// TIA Portal V17 export
// export: Created 2022-07-28T18:03:17.6934733Z, ExportSetting None, DisplayName Totally Integrated Automation Portal, DisplayVersion V17, DisplayName TIA Portal Openness, DisplayVersion V17, DisplayName TIA Portal Teamcenter Gateway, DisplayVersion V17, DisplayName TIA Portal Version Control Interface, DisplayVersion V17, DisplayName TIA Portal Test Suite Advanced, DisplayVersion V17, DisplayName SINAMICS Startdrive Advanced, DisplayVersion V17, DisplayName SINAMICS DCC, DisplayVersion V17, DisplayName SINAMICS Startdrive G130, G150, S120, S150, SINAMICS MV, S210, DisplayVersion V17, DisplayName SINAMICS Startdrive G110M, G120, G120C, G120D, G120P, G115D, DisplayVersion V17, DisplayName STEP 7 Professional, DisplayVersion V17, DisplayName SIMATIC Energy Suite, DisplayVersion V17, DisplayName STEP 7 CFC, DisplayVersion V17, DisplayName STEP 7 Safety, DisplayVersion V17, DisplayName WinCC Advanced / Unified PC, DisplayVersion V17, DisplayName SIMATIC Visualization Architect, DisplayVersion V17
TYPE "Lib_UDT_Int"
   STRUCT
      Tmp : Bool;   // Temp bool Var
      i_Tmp : Int;   // Temp Int Var
      r_Tmp : Real;   // Temp Real Var
      w_Tmp : Word;   // Temp Word Var
      dw_Tmp : DWord;   // Temp Dword Var
      di_Tmp : DInt;   // Temp DInt Var
      AlwTrue : Bool := true;   // Always = True
      AlwFalse : Bool;   // Always = False
      i_Alw0 : Int;   // Always = 0
      b_Alw0 : Byte;   // Always = b#16#0
      w_Alw0 : Word;   // Always = w#16#0
      d_Alw0 : DWord;   // Always = dw#16#0
   END_STRUCT;
END_TYPE
